// TIA Portal V15.1 export
// export: Created 2020-06-12T07:35:42.3505859Z, ExportSetting None, DisplayName Totally Integrated Automation Portal, DisplayVersion V15.1, DisplayName TIA Portal Openness, DisplayVersion V15.1, DisplayName STEP 7 Professional, DisplayVersion V15.1, DisplayName STEP 7 Safety, DisplayVersion V15.1, DisplayName WinCC Advanced, DisplayVersion V15.1
FUNCTION "ES1Sx_io" : Void   // FC137, FBD
{ S7_Optimized_Access := 'TRUE' }
// stored: SetENOAutomatically False
BEGIN

REGION Network 1
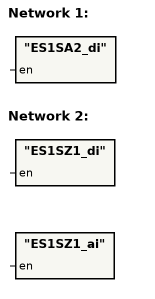
   "ES1SA2_di"();
END_REGION

REGION Network 2
   "ES1SZ1_di"();
   "ES1SZ1_ai"();
END_REGION
END_FUNCTION
